Universal Robots PolyScope program: cobotique capot 3.2.urp

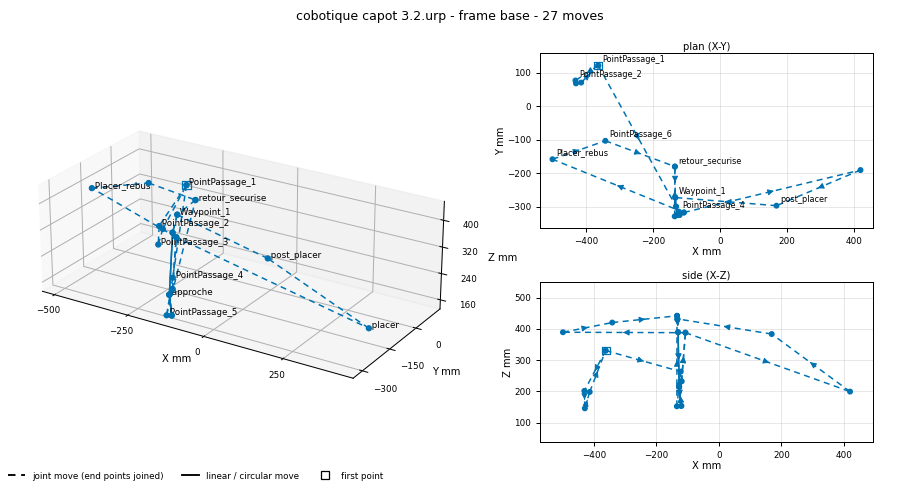
[picture p0: tool path of cobotique capot 3.2.urp in frame base, 27 of 27 moves have a stored position in this frame; points joined in program order, loops and branches not executed]
Program cobotique capot 4 (installation=default directory=/programs/nouveau dossier createdIn=5.8.0.10253 lastSavedIn=5.8.0.10253 robotSerialNumber=20205300713)
Calibrated DH parameters: a=[-0.000115, -0.234909, -0.179769, -0.000009, 0.000011, 0]; d=[0.152009, 9.56008, 250.062401, -259.491708, 0.085429, 0.092054]; alpha=[1.570407, -0.006797, 0.000443, 1.572497, -1.571849, 0]; deltaTheta=[0, -0.26984, 0.838992, -0.569138, 0.000025, 0]
Robot Program (runOnlyOnce=false)
  URCap Activer la main (Robotiq_Grippers, Robotiq Inc.) dataModel(ResetAndActivateKey=false)
  URCap Main (Robotiq_Grippers, Robotiq Inc.) dataModel(position=0.0, force=100.0, speed=100.0, positionInDouble=0.0, forceInDouble=100.0, speedInDouble=100.0, slaveIds=[9], blocking=true)
  URCap Dorner Conveyor (DornerConveyor, Advanced Motion - Controls) dataModel(conv=1, oper=4)
  MoveJ speed 60 deg/s, acceleration 80 deg/s^2 (useActiveTCP=true) feature=Base
    Waypoint PointPassage_1: TCP in base x=-362.873 y=121.551 z=330.941 mm, rx=-1.9188 ry=1.9619 rz=-0.4861 rad; joints [-178.788, -125.505, -25.728, -147.197, 90.384, -177.225] deg
    Waypoint PointPassage_2: TCP in base x=-430.97 y=76.894 z=201.714 mm, rx=2.0698 ry=-2.0943 rz=-0.1905 rad; joints [-173.149, -119.805, -85.495, -51.463, 90.588, -172.064] deg
    Waypoint PointPassage_3: TCP in base x=-429.322 y=68.204 z=145.924 mm, rx=1.8805 ry=-1.9322 rz=-0.5309 rad; joints [-170.647, -128.673, -100.61, -9.403, 84.827, -170.288] deg
    URCap Main (Robotiq_Grippers, Robotiq Inc.) dataModel(position=58.431372549019606, force=100.0, speed=0.0, positionInDouble=58.431372549019606, forceInDouble=100.0, speedInDouble=0.0, slaveIds=[9], blocking=true)
    Waypoint PointPassage_7: TCP in base x=-413.817 y=70.662 z=198.378 mm, rx=1.9115 ry=-1.9576 rz=-0.5039 rad; joints [-170.653, -116.684, -101.489, -22.912, 84.838, -170.288] deg
    Waypoint PointPassage_1: TCP in base x=-362.873 y=121.551 z=330.941 mm, rx=-1.9188 ry=1.9619 rz=-0.4861 rad; joints [-178.788, -125.505, -25.728, -147.197, 90.384, -177.225] deg
    Waypoint PointPassage_4: TCP in base x=-122.288 y=-314.514 z=263.533 mm, rx=3.0821 ry=-0.0339 rz=0.0158 rad; joints [-88.947, -92.859, -99.316, -74.353, 90.389, -177.22] deg
    Waypoint PointPassage_5: motionParameters(jointSpeed=1.047198 jointAcceleration=0.523599 cartesianSpeed=0.25 cartesianAcceleration=1.2); TCP in base x=-134.793 y=-328.518 z=152.429 mm, rx=-2.2052 ry=2.2089 rz=-0.051 rad; joints [-91.616, -109.7, -110.395, -49.373, 91.965, -91.089] deg
    URCap Main (Robotiq_Grippers, Robotiq Inc.) dataModel(position=0.0, force=0.0, speed=0.0, positionInDouble=0.0, forceInDouble=0.0, speedInDouble=0.0, slaveIds=[9], blocking=true)
    Waypoint retour_securise: TCP in base x=-134.176 y=-179.969 z=442.128 mm, rx=-2.2471 ry=-2.1697 rz=0.0496 rad; joints [-90.577, -75.287, -61.755, -132.356, 88.017, -268.12] deg
  Wait Condition expression=digital_in[4] ≟ True  or digital_in[5]≟ True
  If digital_in[4]≟ True
    var_1 := True
    Loop While (checkContinuously=false) expression=var_1≟ True
      MoveJ speed 60 deg/s, acceleration 80 deg/s^2 (useActiveTCP=true) feature=Base
        Waypoint Waypoint_1: TCP in base x=-133.008 y=-272.418 z=432.243 mm, rx=-3.0225 ry=-0.0332 rz=-0.2288 rad; joints [-93.401, -100.875, -37.472, -138.494, 98.06, -184.708] deg
      MoveJ speed 60 deg/s, acceleration 80 deg/s^2 (useActiveTCP=true) feature=Base
        Waypoint photo: TCP in base x=-130.985 y=-299.302 z=389.59 mm, rx=-2.5837 ry=-0.1772 rz=-0.0772 rad; joints [-90.403, -121.375, -12.745, -167.534, 90.797, -188.063] deg
